// Mitsubishi GX Works2 project: may_dap   PLC: FX3S

PROGRAM MAIN
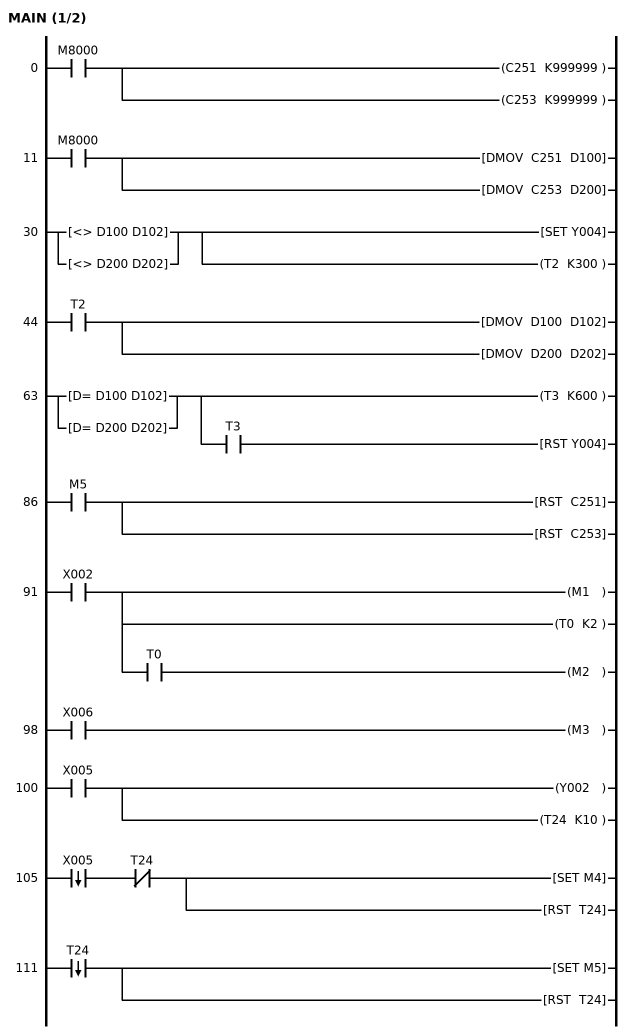
0     LD      M8000
      OUT     C251 K999999
      OUT     C253 K999999
11    LD      M8000
      DMOV    C251 D100
      DMOV    C253 D200
30    LD<>    D100 D102
      OR<>    D200 D202
      SET     Y004
      OUT     T2 K300
44    LD      T2
      DMOV    D100 D102
      DMOV    D200 D202
63    LDD=    D100 D102
      ORD=    D200 D202
      OUT     T3 K600
      AND     T3
      RST     Y004
86    LD      M5
      RST     C251
      RST     C253
91    LD      X002
      OUT     M1
      OUT     T0 K2
      AND     T0
      OUT     M2
98    LD      X006
      OUT     M3
100   LD      X005
      OUT     Y002
      OUT     T24 K10
105   LDF     X005
      ANI     T24
      SET     M4
      RST     T24
111   LDF     T24
      SET     M5
      RST     T24
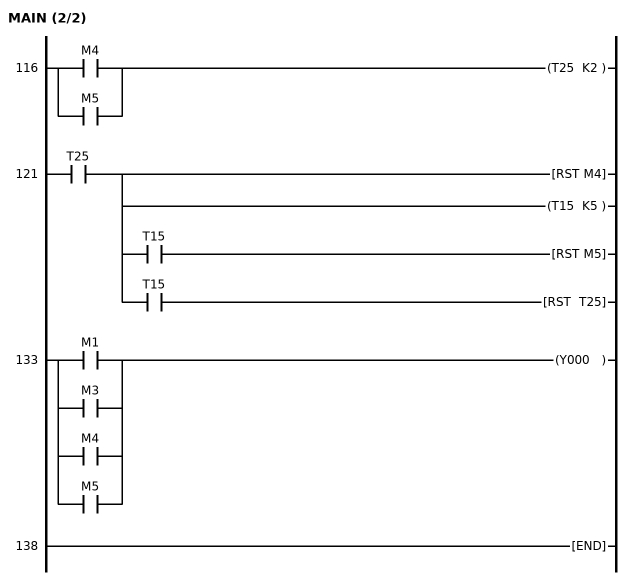
116   LD      M4
      OR      M5
      OUT     T25 K2
121   LD      T25
      RST     M4
      OUT     T15 K5
      MPS
      AND     T15
      RST     M5
      MPP
      AND     T15
      RST     T25
133   LD      M1
      OR      M3
      OR      M4
      OR      M5
      OUT     Y000
138   END
END_PROGRAM
